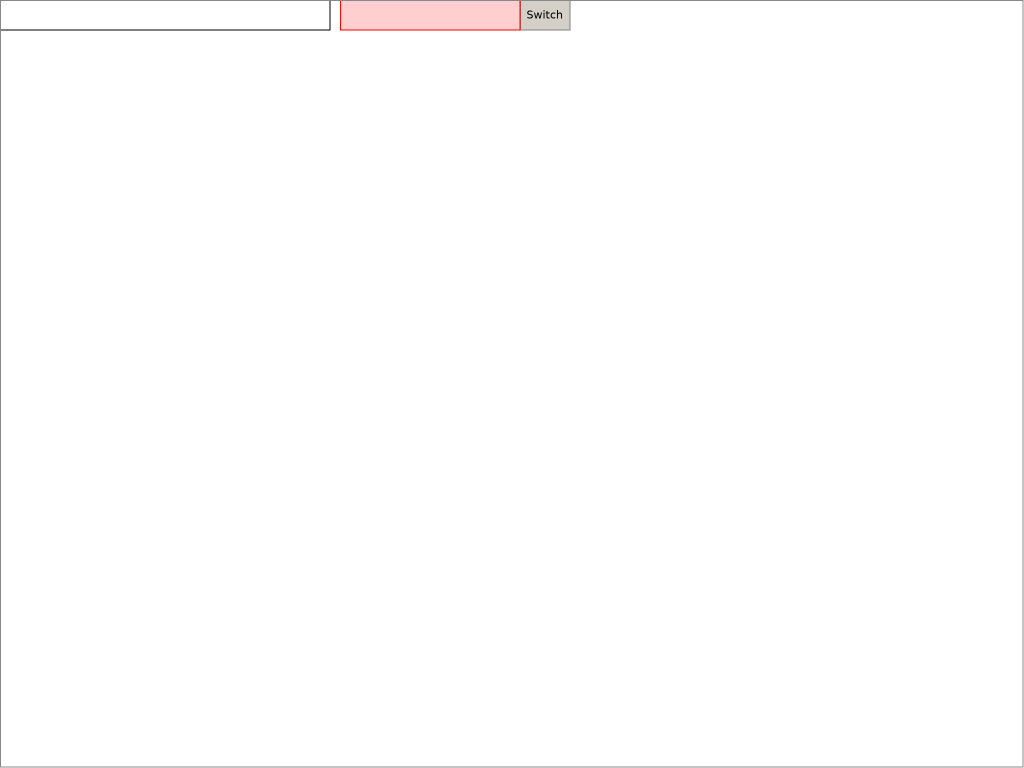
VISUALIZATION Param_BOOL  // 1024x768
VAR_INPUT
	nIdx:		INT;
END_VAR
    Rectangle (0,0 330x30), text list: 'TL_Params_BOOL', text index: nIdx
    Rectangle (520,0 50x30), "Switch", colour toggle: stMParam_Visu.bBoolSetValue[nIdx]
        OnMouseClick: execute { stMParam_Visu.bBoolSetValue[nIdx]:=TRUE; }
    Rectangle (340,0 180x30), colour toggle: stMParam_Visu.bBoolAktValue[nIdx]
    Rectangle (600,0 150x30)
END_VISUALIZATION

(* stored: Version 1.1.0.1
   Visu Param_BOOL: Id {6a9fec63-707b-4079-8363-d50e362b6c13} *)
